Fanuc KAREL source: kt00489.KL

-- PROVISIONAL review KL for V940-1; original PC SHA256 ea1f887098746ff1a03a82c4c469bfd054835e8ae3cb6b11287e365821428ca3
-- Incomplete behavior may be omitted. Consult companion uncertainty JSON. Do not deploy.
PROGRAM KT00489
%NOLOCKGROUP
-- UNRESOLVED_DECL P1 type=000101
-- UNRESOLVED_DECL P2 type=000199
-- UNRESOLVED_DECL OUT type=000101
BEGIN
  -- V9_ZERO_TABLE_METADATA_HINT layout=0001; no indexed target words; source/name/runtime held
  -- UNRESOLVED_PC offsets 5-34; opcodes 49,49,7E,60,4A
  -- UNRESOLVED_PC offsets 39-43; opcodes 7F
END KT00489
